// Mitsubishi GX Works2 project: NIAP1856_1000_CC-1M_R3   PLC: FX3S

PROGRAM MAIN
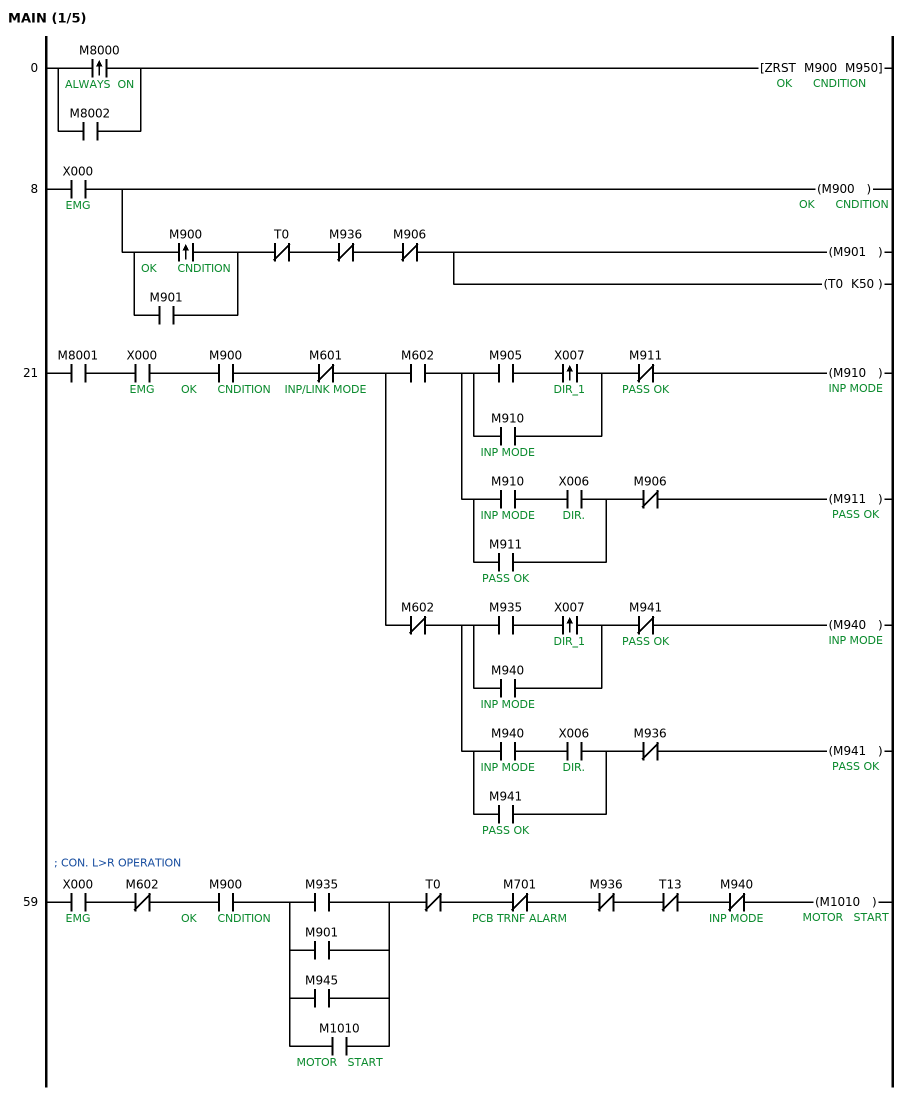
0     LDP     M8000  ; ALWAYS  ON
      OR      M8002
      ZRST    M900 M950  ; OK      CNDITION
8     LD      X000  ; EMG
      OUT     M900  ; OK      CNDITION
      LDP     M900  ; OK      CNDITION
      OR      M901
      ANB
      ANI     T0
      ANI     M936
      ANI     M906
      OUT     M901
      OUT     T0 K50
21    LD      M8001
      AND     X000  ; EMG
      AND     M900  ; OK      CNDITION
      ANI     M601  ; INP/LINK MODE
      MPS
      AND     M602
      MPS
      LD      M905
      ANDP    X007  ; DIR_1
      OR      M910  ; INP MODE
      ANB
      ANI     M911  ; PASS OK
      OUT     M910  ; INP MODE
      MPP
      LD      M910  ; INP MODE
      AND     X006  ; DIR.
      OR      M911  ; PASS OK
      ANB
      ANI     M906
      OUT     M911  ; PASS OK
      MPP
      ANI     M602
      MPS
      LD      M935
      ANDP    X007  ; DIR_1
      OR      M940  ; INP MODE
      ANB
      ANI     M941  ; PASS OK
      OUT     M940  ; INP MODE
      MPP
      LD      M940  ; INP MODE
      AND     X006  ; DIR.
      OR      M941  ; PASS OK
      ANB
      ANI     M936
      OUT     M941  ; PASS OK
; CON. L>R OPERATION
59    LD      X000  ; EMG
      ANI     M602
      AND     M900  ; OK      CNDITION
      LD      M935
      OR      M901
      OR      M945
      OR      M1010  ; MOTOR   START
      ANB
      ANI     T0
      ANI     M701  ; PCB TRNF ALARM
      ANI     M936
      ANI     T13
      ANI     M940  ; INP MODE
      OUT     M1010  ; MOTOR   START
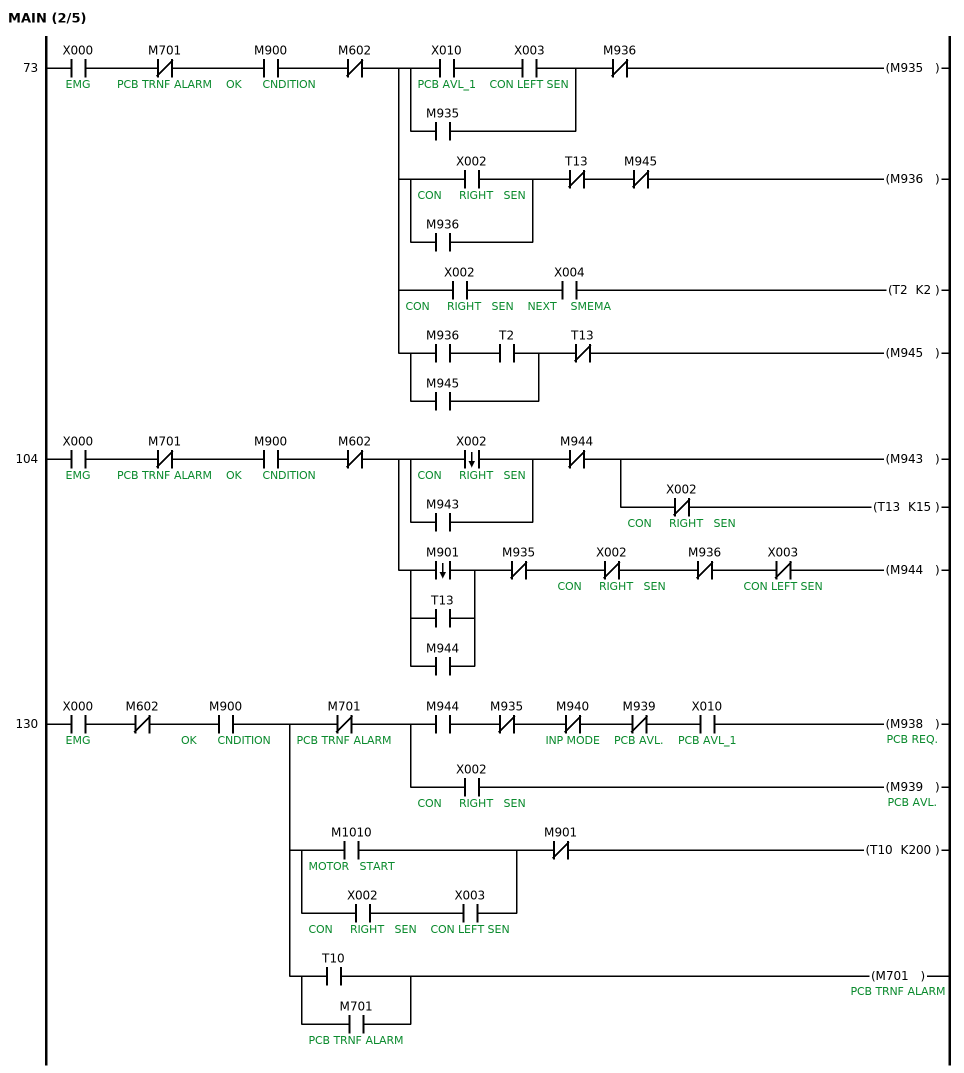
73    LD      X000  ; EMG
      ANI     M701  ; PCB TRNF ALARM
      AND     M900  ; OK      CNDITION
      ANI     M602
      MPS
      LD      X010  ; PCB AVL_1
      AND     X003  ; CON LEFT SEN
      OR      M935
      ANB
      ANI     M936
      OUT     M935
      MRD
      LD      X002  ; CON     RIGHT   SEN
      OR      M936
      ANB
      ANI     T13
      ANI     M945
      OUT     M936
      MRD
      AND     X002  ; CON     RIGHT   SEN
      AND     X004  ; NEXT    SMEMA
      OUT     T2 K2
      MPP
      LD      M936
      AND     T2
      OR      M945
      ANB
      ANI     T13
      OUT     M945
104   LD      X000  ; EMG
      ANI     M701  ; PCB TRNF ALARM
      AND     M900  ; OK      CNDITION
      ANI     M602
      MPS
      LDF     X002  ; CON     RIGHT   SEN
      OR      M943
      ANB
      ANI     M944
      OUT     M943
      ANI     X002  ; CON     RIGHT   SEN
      OUT     T13 K15
      MPP
      LDF     M901
      OR      T13
      OR      M944
      ANB
      ANI     M935
      ANI     X002  ; CON     RIGHT   SEN
      ANI     M936
      ANI     X003  ; CON LEFT SEN
      OUT     M944
130   LD      X000  ; EMG
      ANI     M602
      AND     M900  ; OK      CNDITION
      MPS
      ANI     M701  ; PCB TRNF ALARM
      MPS
      AND     M944
      ANI     M935
      ANI     M940  ; INP MODE
      ANI     M939  ; PCB AVL.
      AND     X010  ; PCB AVL_1
      OUT     M938  ; PCB REQ.
      MPP
      AND     X002  ; CON     RIGHT   SEN
      OUT     M939  ; PCB AVL.
      MRD
      LD      M1010  ; MOTOR   START
      LD      X002  ; CON     RIGHT   SEN
      AND     X003  ; CON LEFT SEN
      ORB
      ANB
      ANI     M901
      OUT     T10 K200
      MPP
      LD      T10
      OR      M701  ; PCB TRNF ALARM
      ANB
      OUT     M701  ; PCB TRNF ALARM
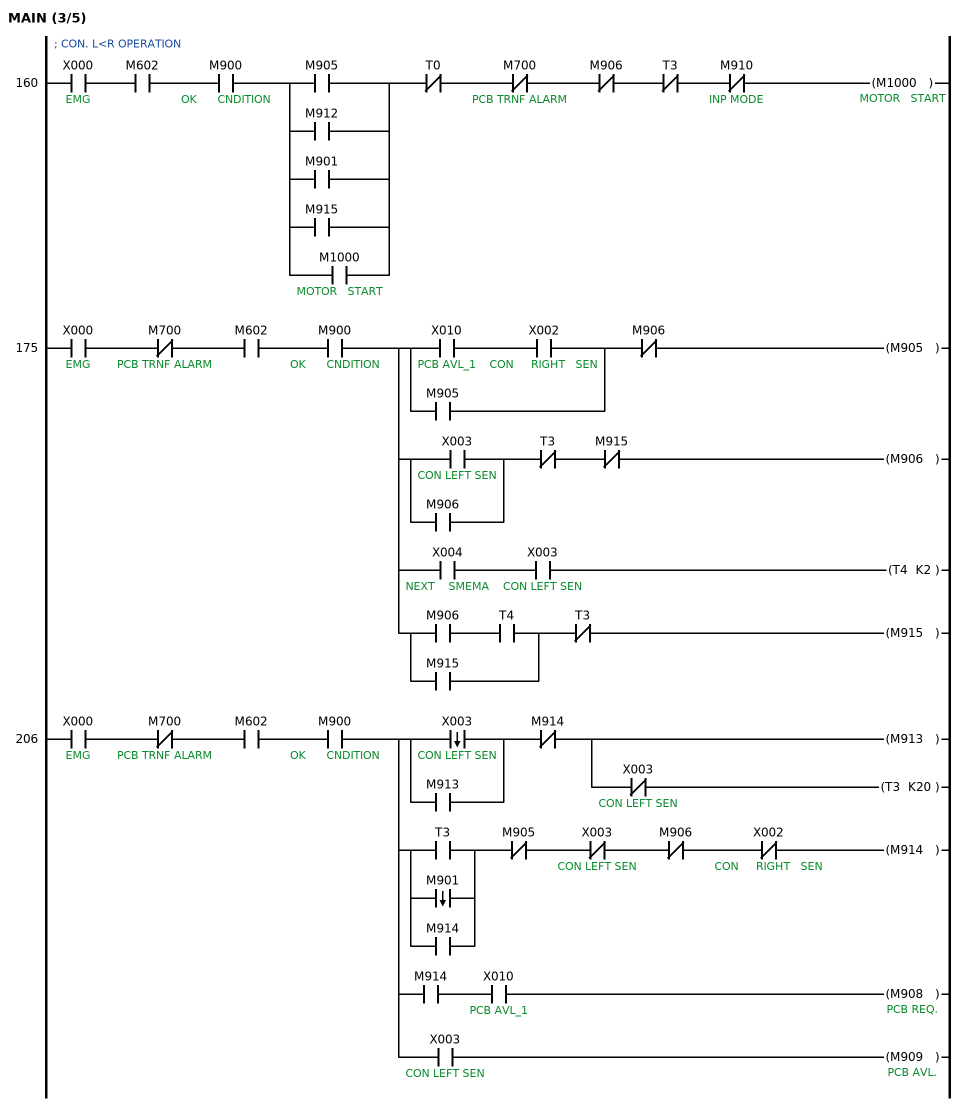
; CON. L<R OPERATION
160   LD      X000  ; EMG
      AND     M602
      AND     M900  ; OK      CNDITION
      LD      M905
      OR      M912
      OR      M901
      OR      M915
      OR      M1000  ; MOTOR   START
      ANB
      ANI     T0
      ANI     M700  ; PCB TRNF ALARM
      ANI     M906
      ANI     T3
      ANI     M910  ; INP MODE
      OUT     M1000  ; MOTOR   START
175   LD      X000  ; EMG
      ANI     M700  ; PCB TRNF ALARM
      AND     M602
      AND     M900  ; OK      CNDITION
      MPS
      LD      X010  ; PCB AVL_1
      AND     X002  ; CON     RIGHT   SEN
      OR      M905
      ANB
      ANI     M906
      OUT     M905
      MRD
      LD      X003  ; CON LEFT SEN
      OR      M906
      ANB
      ANI     T3
      ANI     M915
      OUT     M906
      MRD
      AND     X004  ; NEXT    SMEMA
      AND     X003  ; CON LEFT SEN
      OUT     T4 K2
      MPP
      LD      M906
      AND     T4
      OR      M915
      ANB
      ANI     T3
      OUT     M915
206   LD      X000  ; EMG
      ANI     M700  ; PCB TRNF ALARM
      AND     M602
      AND     M900  ; OK      CNDITION
      MPS
      LDF     X003  ; CON LEFT SEN
      OR      M913
      ANB
      ANI     M914
      OUT     M913
      ANI     X003  ; CON LEFT SEN
      OUT     T3 K20
      MRD
      LD      T3
      ORF     M901
      OR      M914
      ANB
      ANI     M905
      ANI     X003  ; CON LEFT SEN
      ANI     M906
      ANI     X002  ; CON     RIGHT   SEN
      OUT     M914
      MRD
      AND     M914
      AND     X010  ; PCB AVL_1
      OUT     M908  ; PCB REQ.
      MPP
      AND     X003  ; CON LEFT SEN
      OUT     M909  ; PCB AVL.
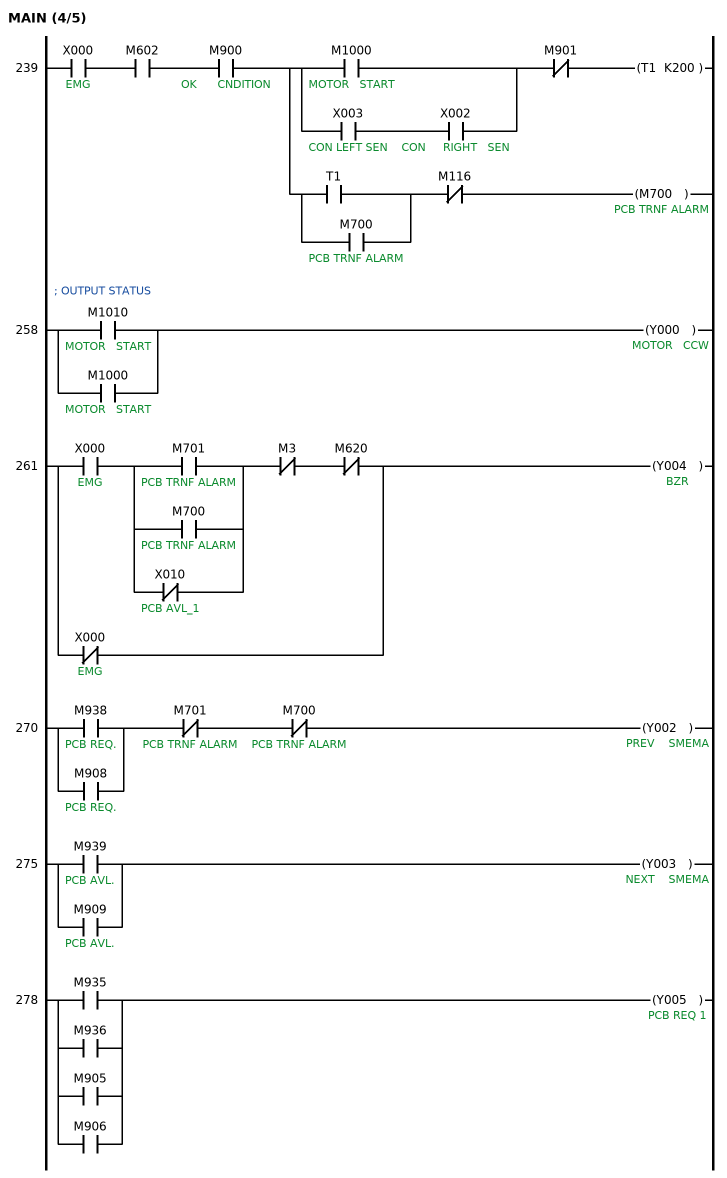
239   LD      X000  ; EMG
      AND     M602
      AND     M900  ; OK      CNDITION
      MPS
      LD      M1000  ; MOTOR   START
      LD      X003  ; CON LEFT SEN
      AND     X002  ; CON     RIGHT   SEN
      ORB
      ANB
      ANI     M901
      OUT     T1 K200
      MPP
      LD      T1
      OR      M700  ; PCB TRNF ALARM
      ANB
      ANI     M116
      OUT     M700  ; PCB TRNF ALARM
; OUTPUT STATUS
258   LD      M1010  ; MOTOR   START
      OR      M1000  ; MOTOR   START
      OUT     Y000  ; MOTOR   CCW
261   LD      X000  ; EMG
      LD      M701  ; PCB TRNF ALARM
      OR      M700  ; PCB TRNF ALARM
      ORI     X010  ; PCB AVL_1
      ANB
      ANI     M3
      ANI     M620
      ORI     X000  ; EMG
      OUT     Y004  ; BZR
270   LD      M938  ; PCB REQ.
      OR      M908  ; PCB REQ.
      ANI     M701  ; PCB TRNF ALARM
      ANI     M700  ; PCB TRNF ALARM
      OUT     Y002  ; PREV    SMEMA
275   LD      M939  ; PCB AVL.
      OR      M909  ; PCB AVL.
      OUT     Y003  ; NEXT    SMEMA
278   LD      M935
      OR      M936
      OR      M905
      OR      M906
      OUT     Y005  ; PCB REQ 1
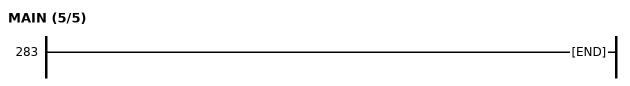
283   END
END_PROGRAM

// device comments not shown above
X001  ; RESET PB
X005  ; PREV    SMEMA
X011  ; PCB REQ_2
X012  ; PCB AVL_2
X015  ; DIRETION
M1  ; HMI     START
M15  ; HMI PASS
M16  ; HMI     RESET
M20  ; HMI     CALIB
M26  ; INTRPD  SIGNAL
M27  ; PRO     COUNT
M44  ; CONVEYOR HOME
M67  ; PRO     CHANGE
M94  ; MANUAL  MODE
M99  ; MOV TRCK ALARM
M102  ; HOME GO TGR
M500  ; HMI     CONFIRM
M600  ; L<R/L>R
M902  ; PCB SEND
M903  ; PCB NOT SEND
M932  ; PCB SEND
M933  ; PCB NOT SEND
M1215  ; HMI CUNT RESET
M1216  ; COUNT   EQUAL
M1310  ; HMI     LOGIN
M1315  ; ACCESS  OK
M1316  ; HMI     LOGOUT
M1320  ; OPT OK
M1330  ; MNT OK
M1340  ; ENG OK
D798  ; PRO     COUNT
D799  ; SET     COUNT
D998  ; HMI     SCREEN
D1000  ; WIDTH   POSITION
D1004  ; CONVEYOR SPEED
D1022  ; WIDTH   COUNT
Y001  ; MOTOR   CW
Y006  ; PASS PB IND
Y007  ; PCB REQ 2
Y010  ; PCB AVL 2
